// TIA Portal V19 export
TYPE "type_u3ResponsetData"
// stored: Access Published, Namespace Unit3
   STRUCT
      u1XyzToU3Tansfered : Bool;   // 是否允许运动
      u2XyzToU3Tansfered : Bool;   // 是否允许运动
   END_STRUCT;
END_TYPE
